{attribute 'qualified_only'}
{attribute 'strict'}
TYPE EBeamShaingFlow :
(
	HS := 0,
	HT
);
END_TYPE

(* stored: Version 1.1.0.1, ProductVersion 3.1.4024.3
   DUT EBeamShaingFlow: Id {6dae7073-3b07-4627-9870-024cc0619955} *)
